FUNCTION_BLOCK SludgeBufferActuators_2 (* Composite Function Block Type *)
  (* Standard: 61499-2 *)
  (* Version 1.0, 9/30/2026, Claude/Hidryco, Schneider Electric, Rev1 - Intertravamentos Pump3/ValveInfeed destrocados *)
  PACKAGE SE.Nereda;
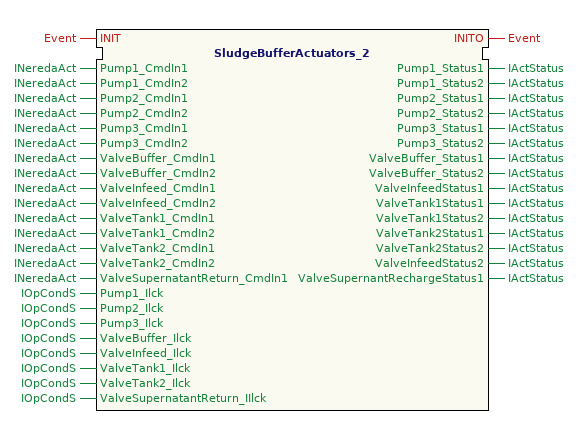
  EVENT_INPUT
    INIT;
  END_EVENT
  EVENT_OUTPUT
    INITO;
  END_EVENT
  SOCKETS
    Pump1_CmdIn1 : INeredaAct;
    Pump1_CmdIn2 : INeredaAct;
    Pump2_CmdIn1 : INeredaAct;
    Pump2_CmdIn2 : INeredaAct;
    Pump3_CmdIn1 : INeredaAct;
    Pump3_CmdIn2 : INeredaAct;
    ValveBuffer_CmdIn1 : INeredaAct;
    ValveBuffer_CmdIn2 : INeredaAct;
    ValveInfeed_CmdIn1 : INeredaAct;
    ValveInfeed_CmdIn2 : INeredaAct;
    ValveTank1_CmdIn1 : INeredaAct;
    ValveTank1_CmdIn2 : INeredaAct;
    ValveTank2_CmdIn1 : INeredaAct;
    ValveTank2_CmdIn2 : INeredaAct;
    ValveSupernatantReturn_CmdIn1 : INeredaAct;
    Pump1_Ilck : IOpCondS; (* Condition summary chain input from upstream blocks *)
    Pump2_Ilck : IOpCondS; (* Condition summary chain input from upstream blocks *)
    Pump3_Ilck : IOpCondS; (* Condition summary chain input from upstream blocks *)
    ValveBuffer_Ilck : IOpCondS; (* Condition summary chain input from upstream blocks *)
    ValveInfeed_Ilck : IOpCondS; (* Condition summary chain input from upstream blocks *)
    ValveTank1_Ilck : IOpCondS; (* Condition summary chain input from upstream blocks *)
    ValveTank2_Ilck : IOpCondS; (* Condition summary chain input from upstream blocks *)
    ValveSupernatantReturn_IIlck : IOpCondS; (* Condition summary chain input from upstream blocks *)
  END_SOCKETS
  PLUGS
    Pump1_Status1 : IActStatus;
    Pump1_Status2 : IActStatus;
    Pump2_Status1 : IActStatus;
    Pump2_Status2 : IActStatus;
    Pump3_Status1 : IActStatus;
    Pump3_Status2 : IActStatus;
    ValveBuffer_Status1 : IActStatus;
    ValveBuffer_Status2 : IActStatus;
    ValveInfeedStatus1 : IActStatus;
    ValveTank1Status1 : IActStatus;
    ValveTank1Status2 : IActStatus;
    ValveTank2Status1 : IActStatus;
    ValveTank2Status2 : IActStatus;
    ValveInfeedStatus2 : IActStatus;
    ValveSupernantRechargeStatus1 : IActStatus;
  END_PLUGS
  (* 01 - FUNCTIONNAL INPUT INTERFACE *)
  (* 00 - INITIALIZATION *)
  (* 05 - LOGIC *)
  (* 06 - HMI INTERFACE *)
  (* 03 - FIELD INTERFACE *)
  (* 02 - FUNCTIONNAL OUTPUT INTERFACE *)
  (* Actuators Status *)
  (* 04 - CHILDREN *)
  (* 4A - TYPICALS *)
  (* Actuators Command *)
  (* Reset All Actuators *)
  FBS
    ResetAllValves : ResetValvesManager;
    ValveBuffer : ValveS;
    Pump1_Status : MultiActStatus;
    Pump2_Status : MultiActStatus;
    Pump3_Status : MultiActStatus;
    Pump1_Cmd : MultiNeredaCmd;
    Pump2_Cmd : MultiNeredaCmd;
    Pump3_Cmd : MultiNeredaCmd;
    Pump1 : Motor_VS;
    Pump2 : Motor_VS;
    Pump3 : Motor_VS;
    ValveInfeed : ValveS;
    ValveTank1 : ValveS;
    BufferValve_Status1 : MultiActStatus;
    InfeedValve_Status : MultiActStatus;
    ValveTank1_Status : MultiActStatus;
    BufferValve_Cmd1 : MultiNeredaCmd;
    InfeedValve_Cmd1 : MultiNeredaCmd;
    ValveTank1_Cmd1 : MultiNeredaCmd;
    ValveTank2 : ValveS;
    ValveTank2_Status : MultiActStatus;
    ValveTank2_Cmd : MultiNeredaCmd;
    ValveSupernatantReturn : ValveS;
    ValveSupernatantReturn_Status : MultiActStatus;
    ValveSupernatantReturn_Cmd : MultiNeredaCmd;
  END_FBS
  EVENT_CONNECTIONS
    INIT TO ResetAllValves.INIT;
    ResetAllValves.INITO TO INITO;
  END_CONNECTIONS
  ADAPTER_CONNECTIONS
    ValveBuffer.E9B1CB906EB3FD07 TO BufferValve_Status1.18836B5B646921E0;
    BufferValve_Cmd1.30D463C0CF465CCB TO ValveBuffer.476D0447CF6D114C;
    ValveBuffer_Ilck TO ValveBuffer.9C9EE774F196CD99;
    Pump1_Ilck TO Pump1.9C9EE774F196CD99;
    Pump2_Ilck TO Pump2.9C9EE774F196CD99;
    Pump3_Ilck TO Pump3.9C9EE774F196CD99;
    ValveInfeed_Ilck TO ValveInfeed.9C9EE774F196CD99;
    ValveTank1_Ilck TO ValveTank1.9C9EE774F196CD99;
    Pump1_Cmd.30D463C0CF465CCB TO Pump1.D01B7CFFEEA98E7A;
    Pump2_Cmd.30D463C0CF465CCB TO Pump2.D01B7CFFEEA98E7A;
    Pump3_Cmd.30D463C0CF465CCB TO Pump3.D01B7CFFEEA98E7A;
    InfeedValve_Cmd1.30D463C0CF465CCB TO ValveInfeed.476D0447CF6D114C;
    ValveTank1_Cmd1.30D463C0CF465CCB TO ValveTank1.476D0447CF6D114C;
    ValveTank1.E9B1CB906EB3FD07 TO ValveTank1_Status.18836B5B646921E0;
    ValveInfeed.E9B1CB906EB3FD07 TO InfeedValve_Status.18836B5B646921E0;
    Pump2.378A5C96F2B54F0C TO Pump2_Status.18836B5B646921E0;
    Pump3.378A5C96F2B54F0C TO Pump3_Status.18836B5B646921E0;
    Pump1.378A5C96F2B54F0C TO Pump1_Status.18836B5B646921E0;
    Pump1_CmdIn1 TO Pump1_Cmd.F1CE5E5BC0F88348;
    Pump1_CmdIn2 TO Pump1_Cmd.814FBE7646911966;
    Pump2_CmdIn1 TO Pump2_Cmd.F1CE5E5BC0F88348;
    Pump2_CmdIn2 TO Pump2_Cmd.814FBE7646911966;
    Pump3_CmdIn1 TO Pump3_Cmd.F1CE5E5BC0F88348;
    Pump3_CmdIn2 TO Pump3_Cmd.814FBE7646911966;
    ValveBuffer_CmdIn1 TO BufferValve_Cmd1.F1CE5E5BC0F88348;
    ValveBuffer_CmdIn2 TO BufferValve_Cmd1.814FBE7646911966;
    ValveInfeed_CmdIn1 TO InfeedValve_Cmd1.F1CE5E5BC0F88348;
    ValveInfeed_CmdIn2 TO InfeedValve_Cmd1.814FBE7646911966;
    ValveTank1_CmdIn1 TO ValveTank1_Cmd1.F1CE5E5BC0F88348;
    ValveTank1_CmdIn2 TO ValveTank1_Cmd1.814FBE7646911966;
    ResetAllValves.2 TO ValveBuffer.76FFF418213BE03C;
    ResetAllValves.5 TO ValveInfeed.76FFF418213BE03C;
    ResetAllValves.6 TO ValveTank1.76FFF418213BE03C;
    ValveTank2_Cmd.30D463C0CF465CCB TO ValveTank2.476D0447CF6D114C;
    ValveTank2.E9B1CB906EB3FD07 TO ValveTank2_Status.18836B5B646921E0;
    ValveTank2_Ilck TO ValveTank2.9C9EE774F196CD99;
    ResetAllValves.7 TO ValveTank2.76FFF418213BE03C;
    ValveTank2_CmdIn1 TO ValveTank2_Cmd.F1CE5E5BC0F88348;
    ValveTank2_CmdIn2 TO ValveTank2_Cmd.814FBE7646911966;
    Pump1_Status.8244952938F4EC92 TO Pump1_Status1;
    Pump1_Status.3FD61FA75EE1C84B TO Pump1_Status2;
    Pump2_Status.8244952938F4EC92 TO Pump2_Status1;
    Pump2_Status.3FD61FA75EE1C84B TO Pump2_Status2;
    Pump3_Status.8244952938F4EC92 TO Pump3_Status1;
    Pump3_Status.3FD61FA75EE1C84B TO Pump3_Status2;
    BufferValve_Status1.8244952938F4EC92 TO ValveBuffer_Status1;
    BufferValve_Status1.3FD61FA75EE1C84B TO ValveBuffer_Status2;
    InfeedValve_Status.8244952938F4EC92 TO ValveInfeedStatus1;
    InfeedValve_Status.3FD61FA75EE1C84B TO ValveInfeedStatus2;
    ValveTank1_Status.8244952938F4EC92 TO ValveTank1Status1;
    ValveTank1_Status.3FD61FA75EE1C84B TO ValveTank1Status2;
    ValveTank2_Status.8244952938F4EC92 TO ValveTank2Status1;
    ValveTank2_Status.3FD61FA75EE1C84B TO ValveTank2Status2;
    ValveSupernatantReturn_Cmd.30D463C0CF465CCB TO ValveSupernatantReturn.476D0447CF6D114C;
    ValveSupernatantReturn.E9B1CB906EB3FD07 TO ValveSupernatantReturn_Status.18836B5B646921E0;
    ResetAllValves.8 TO ValveSupernatantReturn.76FFF418213BE03C;
    ValveSupernatantReturn_IIlck TO ValveSupernatantReturn.9C9EE774F196CD99;
    ValveSupernatantReturn_CmdIn1 TO ValveSupernatantReturn_Cmd.F1CE5E5BC0F88348;
    ValveSupernatantReturn_Status.8244952938F4EC92 TO ValveSupernantRechargeStatus1;
  END_CONNECTIONS
END_FUNCTION_BLOCK
